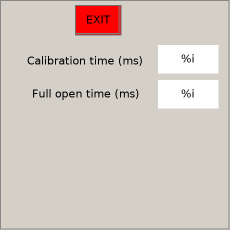
VISUALIZATION ExtractiveOutletValveParameterMenu  // 230x230
    Textfield (157,44 62x30), "%i", text variable: AutoExtractionParameterMenuBindings.refillIntervalTextField_TextVariable
        OnMouseDown: write the text variable via VisuDialogs.Numpad, min 1, max 999
    Label (23,39 124x44), "Calibration time (ms)"
    Button (75,5 46x30), "EXIT", pressed state: NOT MainScreenBindings.autoExtractionParameterMenuButton_ToggleVariable
        toggle MainScreenBindings.ControlValveParameterMenuButton_ToggleVariable
    Textfield (157,79 62x30), "%i", text variable: AutoExtractionParameterMenuBindings.pumpSetpointWaitTimeTextField_TextVariable
        OnMouseDown: write the text variable via VisuDialogs.Numpad, min 0, max 999
    Label (24,72 124x44), "Full open time (ms)"
END_VISUALIZATION

(* stored: Version 1.1.0.1, ProductVersion 3.1.4024.9
   Visu ExtractiveOutletValveParameterMenu: Id {f32f2d73-1832-423e-aa99-56e2bcba349c} *)
